# B&R Automation Studio project GroupProjectBR
Automation Studio 4.12.4.107 SP; Project that includes both HMI visualization and script of controling conveyor belt and sorting system.; technology packages: mappCockpit 5.23.0, mappMotion 5.23.0, mappView 5.23.0

## Configuration ConfigSortingSystem

CPU X20CP1584, AutomationRuntime B4.93, Build 4.1.2, Vc V4.72.6

### Hardware
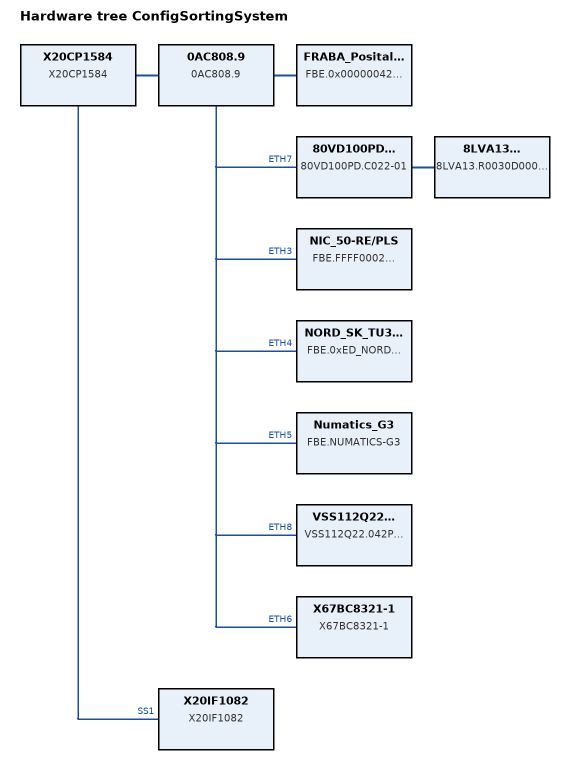
```
0AC808.9 : 0AC808.9 v1.0.0.0  [ETH1 -> X20CP1584.IF3 [Cable Type=PowerlinkCable, Length=10, Version=1.0.0.3]; ETH2 -> FRABA_Posital_Absolute_Rotary_Encoder.PLK1 [Cable Type=PowerlinkCable, Length=10, Version=1.0.0.3]; ETH3 -> NIC_50-RE/PLS.PLK1 [Cable Type=PowerlinkCable, Length=10, Version=1.0.0.3]; ETH4 -> NORD_SK_TU3-POL_SK54xE_Inverter.PLK1 [Cable Type=PowerlinkCable, Length=10, Version=1.0.0.3]; ETH5 -> Numatics_G3.PLK1 [Cable Type=PowerlinkCable, Length=10, Version=1.0.0.3]; ETH6 -> X67BC8321-1.PLK1 [Cable Type=PowerlinkCable, Length=10, Version=1.0.0.3]; ETH7 -> 80VD100PD.C022-01.PLK2 [Cable Type=PowerlinkCable, Length=10, Version=1.0.0.3]; ETH8 -> VSS112Q22.042P-000.PLK1 [Cable Type=PowerlinkCable, Length=10, Version=1.0.0.3]]
80VD100PD.C022-01 : 80VD100PD.C022-01 v2.5.0.0  [PLK2 -> 0AC808.9.ETH7 (NodeNumber=9) [Cable Type=PowerlinkCable, Length=10, Version=1.0.0.3]]
  DriveConfiguration/Module:
    McAcoposTypeID = AcoposMicroDConfig
    ActivateACOPOSSimulationOnPLC = 0
  DriveConfiguration/Encoder/EncoderX6A/InterfaceType:
    ResolverPolepairs = 1
  DriveConfiguration/Encoder/EncoderX6B/InterfaceType:
    ResolverPolepairs = 1
  DriveConfiguration/Channel[1]/RealAxis:
    AxisReference = gAxis_1
    MechanicalElementsIsInvisible = 0
  DriveConfiguration/Channel[1]/RealAxis/MechanicalElements/Gearbox:
    InputIsReadOnly = 0
    Input = 1
    OutputIsReadOnly = 0
    Output = 1
  DriveConfiguration/Channel[1]/RealAxis/MechanicalElements/RotaryToLinearTransformation:
    ReferenceDistanceIsReadOnly = 0
    ReferenceDistance = 175
  DriveConfiguration/Channel[1]/RealAxis/Controller:
    ModeIsReadOnly = 0
    Mode = PositionController
  DriveConfiguration/Channel[1]/RealAxis/Controller/Mode/Position:
    ProportionalGain = 194
    IntegrationTime = 0.0
    PredictionTime = 0.0004
    TotalDelayTime = 0.0004
  DriveConfiguration/Channel[1]/RealAxis/Controller/Mode/Speed:
    ProportionalGainIsReadOnly = 0
    ProportionalGain = 0.75
    IntegrationTimeIsReadOnly = 0
    IntegrationTime = 0.0
    FilterTimeIsReadOnly = 0
    FilterTime = 0.0
  DriveConfiguration/Channel[1]/RealAxis/Controller/Mode/LoopFilters:
    LoopFilterXIsReadOnly = 0
    LoopFilter1 = NotUsed
    LoopFilter2 = NotUsed
    LoopFilter3 = NotUsed
  DriveConfiguration/Channel[1]/RealAxis/Homing:
    ModeIsReadOnly = 0
    Mode = Direct
  DriveConfiguration/Channel[1]/RealAxis/Homing/Mode:
    Position = 0.0
    ReferencePulse = NotUsed
  DriveConfiguration/Channel[1]/RealAxis/Homing:
    RestorePositionVariable = 
  DriveConfiguration/Channel[1]/RealAxis/StopReaction:
    QuickstopIsReadOnly = 0
    Quickstop = DecelerationLimit
    DriveErrorIsReadOnly = 0
    DriveError = DecelerationLimit
  DriveConfiguration/Channel[1]/RealAxis/MovementErrorLimits:
    PositionError = 5
    VelocityErrorMonitoring = Automatic1
  DriveConfiguration/Channel[1]/RealAxis:
    JerkFilterIsReadOnly = 0
    JerkFilter = NotUsed
    ZeroVibrationFilter = NotUsed
  DriveConfiguration/Channel[1]/RealAxis/DigitalInputs/HomingSwitch:
    SourceIsReadOnly = 0
    Source = NotUsed
    Level = High
  DriveConfiguration/Channel[1]/RealAxis/DigitalInputs/PositiveLimitSwitch:
    SourceIsReadOnly = 0
    Source = NotUsed
    Level = High
  DriveConfiguration/Channel[1]/RealAxis/DigitalInputs/NegativeLimitSwitch:
    SourceIsReadOnly = 0
    Source = NotUsed
    Level = High
  DriveConfiguration/Channel[1]/RealAxis/DigitalInputs/Trigger1:
    Source = X2Trigger1
    Level = High
  DriveConfiguration/Channel[1]/RealAxis/DigitalInputs/Trigger2:
    Source = X2Trigger2
    Level = High
  DriveConfiguration/Channel[1]/RealAxis/DigitalInputs/Quickstop:
    Input = Trigger2
  DriveConfiguration/Channel[1]/RealAxis/Simulation:
    SimulationModeOnPLC = SetValueGeneration
    SimulationModeOnACOPOS = NotUsed
  DriveConfiguration/Channel[2]/RealAxis:
    AxisReference = 
    MechanicalElementsIsInvisible = 0
  DriveConfiguration/Channel[2]/RealAxis/MechanicalElements/Gearbox:
    InputIsReadOnly = 0
    Input = 1
    OutputIsReadOnly = 0
    Output = 1
  DriveConfiguration/Channel[2]/RealAxis/MechanicalElements/RotaryToLinearTransformation:
    ReferenceDistanceIsReadOnly = 0
    ReferenceDistance = 1
  DriveConfiguration/Channel[2]/RealAxis/Controller:
    ModeIsReadOnly = 0
    Mode = PositionController
  DriveConfiguration/Channel[2]/RealAxis/Controller/Mode/Position:
    ProportionalGain = 50.0
    IntegrationTime = 0.0
    PredictionTime = 0.0004
    TotalDelayTime = 0.0004
  DriveConfiguration/Channel[2]/RealAxis/Controller/Mode/Speed:
    ProportionalGainIsReadOnly = 0
    ProportionalGain = 2.0
    IntegrationTimeIsReadOnly = 0
    IntegrationTime = 0.0
    FilterTimeIsReadOnly = 0
    FilterTime = 0.0
  DriveConfiguration/Channel[2]/RealAxis/Controller/Mode/LoopFilters:
    LoopFilterXIsReadOnly = 0
    LoopFilter1 = NotUsed
    LoopFilter2 = NotUsed
    LoopFilter3 = NotUsed
  DriveConfiguration/Channel[2]/RealAxis/Homing:
    ModeIsReadOnly = 0
    Mode = Direct
  DriveConfiguration/Channel[2]/RealAxis/Homing/Mode:
    Position = 0.0
    ReferencePulse = NotUsed
  DriveConfiguration/Channel[2]/RealAxis/Homing:
    RestorePositionVariable = 
  DriveConfiguration/Channel[2]/RealAxis/StopReaction:
    QuickstopIsReadOnly = 0
    Quickstop = DecelerationLimit
    DriveErrorIsReadOnly = 0
    DriveError = DecelerationLimit
  DriveConfiguration/Channel[2]/RealAxis/MovementErrorLimits:
    PositionError = 1.0
    VelocityErrorMonitoring = Automatic1
  DriveConfiguration/Channel[2]/RealAxis:
    JerkFilterIsReadOnly = 0
    JerkFilter = NotUsed
    ZeroVibrationFilter = NotUsed
  DriveConfiguration/Channel[2]/RealAxis/DigitalInputs/HomingSwitch:
    SourceIsReadOnly = 0
    Source = NotUsed
    Level = High
  DriveConfiguration/Channel[2]/RealAxis/DigitalInputs/PositiveLimitSwitch:
    SourceIsReadOnly = 0
    Source = NotUsed
    Level = High
  DriveConfiguration/Channel[2]/RealAxis/DigitalInputs/NegativeLimitSwitch:
    SourceIsReadOnly = 0
    Source = NotUsed
    Level = High
  DriveConfiguration/Channel[2]/RealAxis/DigitalInputs/Trigger1:
    Source = X2Trigger1
    Level = High
  DriveConfiguration/Channel[2]/RealAxis/DigitalInputs/Trigger2:
    Source = X2Trigger2
    Level = High
  DriveConfiguration/Channel[2]/RealAxis/DigitalInputs/Quickstop:
    Input = Trigger2
  DriveConfiguration/Channel[2]/RealAxis/Simulation:
    SimulationModeOnPLC = SetValueGeneration
    SimulationModeOnACOPOS = NotUsed
8LVA13.R0030D000-0 : 8LVA13.R0030D000-0 v2.2.0.4  [MT -> 80VD100PD.C022-01.MT1]
  M1/MotorParameters:
    MOTOR_AMB_TEMP_RATED = 40
FRABA_Posital_Absolute_Rotary_Encoder : FBE.0x00000042_PowerlinkRotaryEncoder_OCD_V02-10 v1.0 (OrderNumber=FRABA Posital Absolute Rotary Encoder)  [PLK1 -> 0AC808.9.ETH2 (NodeNumber=8) [Cable Type=PowerlinkCable, Length=10, Version=1.0.0.3]]
  Supervision = off
  p2110_value = 
  p6000_value = 
  p6003_value = 
NIC_50-RE/PLS : FBE.FFFF0002_TLBPOWERLINK v1.0 (OrderNumber=NIC 50-RE/PLS)  [PLK1 -> 0AC808.9.ETH3 (NodeNumber=2) [Cable Type=PowerlinkCable, Length=10, Version=1.0.0.3]]
NORD_SK_TU3-POL_SK54xE_Inverter : FBE.0xED_NORD_TU3_POL_SK54xE_Inverter v1.0 (OrderNumber=NORD SK TU3-POL SK54xE Inverter)  [PLK1 -> 0AC808.9.ETH4 (NodeNumber=3) [Cable Type=PowerlinkCable, Length=10, Version=1.0.0.3]]
Numatics_G3 : FBE.NUMATICS-G3 v1.0 (OrderNumber=Numatics G3)  [PLK1 -> 0AC808.9.ETH5 (NodeNumber=6) [Cable Type=PowerlinkCable, Length=10, Version=1.0.0.3]]
  Supervision = off
VSS112Q22.042P-000 : VSS112Q22.042P-000 v1.7.0.605  [PLK1 -> 0AC808.9.ETH8 (NodeNumber=1) [Cable Type=PowerlinkCable, Length=10, Version=1.0.0.3]]
X20CP1584 : X20CP1584 v1.10.0.0
  Connector IF2:
    ActivateDevice = 1
    ActivateSnmp = 2
  ConfigurationID = Group_Project_BR_ConfigSortingSystem
  TimerDeviceType = EPLX2X
  TimerDevice = X20CP1584.IF3
  TaskClassIdleTime = 2000
  FileDevice1
  FileDeviceName1 = USER
  FileDevicePath1 = USER_PATH
  ActivateOpcUa = 1
  OpcUaInformationModels_PV_Version = 1
X20IF1082 : X20IF1082 v1.12.0.0  [SS -> X20CP1584.SS1]
  Connector IF1:
    EplNatSubnet = 192.168.102.0
X67BC8321-1 : X67BC8321-1 v2.14.0.0  [PLK1 -> 0AC808.9.ETH6 (NodeNumber=5) [Cable Type=PowerlinkCable, Length=10, Version=1.0.0.3]]
```

### IoMap.iom - X20CP1584/IoMap.iom
```iecst
VAR_CONFIG
	::Program:BAIT AT %QW."Numatics_G3".Out01_I3201Out;
END_VAR
```

### Config.mpalarmxcore - X20CP1584/mappServices/Config.mpalarmxcore
```
Element gAlarmXCore (Type=mpalarmxcore)
  mapp.AlarmX.Core.Configuration:
    [0]:
      Name = alarm1
      Message = alarm1 info message
      Behavior = DiscreteValueMonitoring
        Monitoring:
          MonitoredPV = ::ProgramAla:alarm1
          TriggerValues:
            [0] = 1
```

### viComp.visioncomponent - X20CP1584/mappVision/viComp.visioncomponent
```
Element gCamera (Type=visioncomponent)
  VisionApplicationReference = ViAppLogo
```

## Logical view

Binary libraries used (declarations not repeated): operator, runtime, astime, AsIecCon, MpAxis, McAxis, MpBase, McAcpAx, CoTrace, AsZip, FileIO, McBase

### Global.var
```iecst
VAR
	ZmiennaSzymona : USINT;
	ZmiennaGlobalnaBartasa : INT;
	ZmiennaGlobalnaBartasa2 : USINT;
END_VAR
```

### Program Logical/Program

#### Variables.var
```iecst
VAR
	GRt : USINT;
	MotorBeltAxisBasic : MpAxisBasic;
	MotorBeltParType : MpAxisBasicParType;
	BAIT : UINT;
	Wysun : BOOL;
	Moja_zmienna_szymon : BOOL;
END_VAR
```

#### Main.st
```iecst
PROGRAM _INIT

	//Wysun; // testowa zmienna

END_PROGRAM

PROGRAM _CYCLIC
//	IF Wysun THEN  //TESTOWANIE
//		BAIT := 2#0000_0000_0000_0101;
//	ELSE
//		BAIT := 2#0000_0000_0000_0000;
//	END_IF;

	//Fragment kodu odpowiedzialny za inicjalizacjê taœmy
	gAxis_1;
	MotorBeltAxisBasic.MpLink := ADR(gAxis_1);
	MotorBeltAxisBasic.Enable := TRUE;
	MotorBeltAxisBasic.Parameters := ADR(MotorBeltParType);

	//dodany komentarz

	MotorBeltAxisBasic();

END_PROGRAM

PROGRAM _EXIT

END_PROGRAM
```

- Main.st.orig (not shown)

#### Main_BACKUP_283.st
```iecst
PROGRAM _INIT
	//BARTAS
	//BARTAS
	//Wysun; // testowa zmienna

END_PROGRAM

PROGRAM _CYCLIC
<<<<<<< HEAD

	//BARTAS
=======
	//przesuwam program SZY
>>>>>>> MASEGR
//	IF Wysun THEN  //TESTOWANIE
//		BAIT := 2#0000_0000_0000_0101;
//	ELSE
//		BAIT := 2#0000_0000_0000_0000;
//	END_IF;

	//Fragment kodu odpowiedzialny za inicjalizacjê taœmy
	gAxis_1;
	MotorBeltAxisBasic.MpLink := ADR(gAxis_1);
	MotorBeltAxisBasic.Enable := TRUE;
	MotorBeltAxisBasic.Parameters := ADR(MotorBeltParType);
	MotorBeltAxisBasic();

END_PROGRAM

PROGRAM _EXIT

	 	//BARTAS
END_PROGRAM
```

#### Main_BASE_283.st
```iecst
PROGRAM _INIT

	//Wysun; // testowa zmienna
	//komentarz SZYMON
END_PROGRAM

PROGRAM _CYCLIC
	//przesuwam program SZYMON
//	IF Wysun THEN  //TESTOWANIE
//		BAIT := 2#0000_0000_0000_0101;
//	ELSE
//		BAIT := 2#0000_0000_0000_0000;
//	END_IF;

	//Fragment kodu odpowiedzialny za inicjalizacjê taœmy
	gAxis_1;
	MotorBeltAxisBasic.MpLink := ADR(gAxis_1);
	MotorBeltAxisBasic.Enable := TRUE;
	MotorBeltAxisBasic.Parameters := ADR(MotorBeltParType);
	MotorBeltAxisBasic();
	//uwaga coœ tutaj pisze SZYMON

END_PROGRAM

PROGRAM _EXIT

END_PROGRAM
```

#### Main_LOCAL_283.st
```iecst
PROGRAM _INIT
	//BARTAS
	//BARTAS
	//Wysun; // testowa zmienna

END_PROGRAM

PROGRAM _CYCLIC

	//BARTAS
//	IF Wysun THEN  //TESTOWANIE
//		BAIT := 2#0000_0000_0000_0101;
//	ELSE
//		BAIT := 2#0000_0000_0000_0000;
//	END_IF;

	//Fragment kodu odpowiedzialny za inicjalizacjê taœmy
	gAxis_1;
	MotorBeltAxisBasic.MpLink := ADR(gAxis_1);
	MotorBeltAxisBasic.Enable := TRUE;
	MotorBeltAxisBasic.Parameters := ADR(MotorBeltParType);
	MotorBeltAxisBasic();

END_PROGRAM

PROGRAM _EXIT

	 	//BARTAS
END_PROGRAM
```

#### Main_REMOTE_363.st
```iecst
PROGRAM _INIT

	//Wysun; // testowa zmienna
	//komentarz SZYMON
END_PROGRAM

PROGRAM _CYCLIC
	//przesuwam program SZY
//	IF Wysun THEN  //TESTOWANIE
//		BAIT := 2#0000_0000_0000_0101;
//	ELSE
//		BAIT := 2#0000_0000_0000_0000;
//	END_IF;

	//Fragment kodu odpowiedzialny za inicjalizacjê taœmy
	gAxis_1;
	MotorBeltAxisBasic.MpLink := ADR(gAxis_1);
	MotorBeltAxisBasic.Enable := TRUE;
	MotorBeltAxisBasic.Parameters := ADR(MotorBeltParType);
	MotorBeltAxisBasic();
	//uwaga coœ tutaj pisze SZYMON

END_PROGRAM

PROGRAM _EXIT

END_PROGRAM
```

### Program Logical/Program3R4TG

#### Main.st
```iecst
PROGRAM _INIT
	(* Insert code here *)

END_PROGRAM

PROGRAM _CYCLIC
	//MAREK
END_PROGRAM

PROGRAM _EXIT
	//JD

END_PROGRAM
```

### Program Logical/ProgramAlarms

#### Variables.var
```iecst
VAR
	MpAlarmXCore_0 : MpAlarmXCore;
	alarm1 : BOOL;
	Zmienna : BOOL;
END_VAR
```

#### Main.st
```iecst
PROGRAM _INIT
	(* Insert code here *)

END_PROGRAM

PROGRAM _CYCLIC
	(* Insert code here *)
	MpAlarmXCore_0.Enable := TRUE;
	MpAlarmXCore_0.MpLink := ADR(gAlarmXCore);
	MpAlarmXCore_0();
END_PROGRAM

PROGRAM _EXIT
	(* Insert code here *)

END_PROGRAM
```

### Program Logical/ZRODLODRZEWO

#### Variables.var
```iecst
VAR
	UHUHUUU : USINT;
END_VAR
```

#### Main.st
```iecst
PROGRAM _INIT
	(* Insert code here *)

END_PROGRAM

PROGRAM _CYCLIC
	//DKSALLLLLLLLLLLLLLLLLLLLLL

END_PROGRAM

PROGRAM _EXIT
	(* Insert code here *)

END_PROGRAM
```
